TYPE T_AnyBytes : __SYSTEM.AnyType; END_TYPE

(* stored: Version 1.1.0.1
   DUT T_AnyBytes: Id {2908adf1-cbe3-4cd7-bf09-372ce3156095} *)
